// TIA Portal V19 export
TYPE "C501_VAR_SME_TYPIC"
   STRUCT
      MWA { ExternalAccessible := 'False'; ExternalVisible := 'False'; ExternalWritable := 'False'} : USInt;   // Meetwaarde
      OBS { ExternalAccessible := 'False'; ExternalVisible := 'False'; ExternalWritable := 'False'} : USInt;   // Observeerbaarheid
   END_STRUCT;
END_TYPE
